Universal Robots PolyScope program: 20240830usb.urp

Program 20240830usb (installation=20240827 directory=/programs/Demos/usb createdIn=5.13.1 lastSavedIn=5.15.1 robotSerialNumber=20245500285)
Calibrated DH parameters: a=[0.000097, -0.210459, -0.026602, 0.000137, 0.000078, 0]; d=[0.162601, 254.180657, -54.076236, -199.970743, 0.099615, 0.099684]; alpha=[1.569796, -0.001455, 0.001957, 1.570525, -1.571561, 0]; deltaTheta=[0, -1.053331, 8.839472, -1.50296, 0.000002, 0]
InitVariablesNode
Robot Program (runOnlyOnce=false)
  MoveJ speed 60 deg/s, acceleration 80 deg/s^2 (useActiveTCP=true) feature=Base
    Waypoint 路点_2: TCP in base x=378.633 y=-400.967 z=269.032 mm, rx=0.8465 ry=2.3153 rz=-0.4134 rad; joints [111.319, -104.713, 126.879, -151.343, -75.69, 66.743] deg; TCP offset x=-0.17 y=0 z=192.95 mm, rx=0 ry=0 rz=0 rad
  Script: usb = rpc_factory("xmlrpc","http://192.168.1.7:9120/RPC2")
  SuppressedNode
    Script: usb.open()
  SuppressedNode
    Popup Message (haltProgram=false message=Grasp will close... inputType=Text)
  SuppressedNode
    Script: usb.close()
  Script: a=usb.get_target_pose()
  var_3 := p[0,0,0,0,0,0]
  Script: var_3[0] = -a[0]
  Script: var_3[2] = a[2]
  Script: var_3[4] = -a[4]
  Popup Message (haltProgram=false message=Get target pose. inputType=Variable) variable=var_3
  MoveJ speed 60 deg/s, acceleration 80 deg/s^2 (useActiveTCP=true) feature=Base
    Waypoint 路点_1: TCP in base x=381.086 y=-304.22 z=65.94 mm, rx=0 ry=3.0695 rz=-0.001 rad; joints [123.239, -85.086, 121.462, -128.728, -86.621, 33.467] deg; TCP offset x=-0.17 y=0 z=192.95 mm, rx=0 ry=0 rz=0 rad
  MoveJ speed 30 deg/s, acceleration 60 deg/s^2 (useActiveTCP=true) feature=Base
    var_1 := get_actual_tcp_pose()
    var_2 := pose_trans(var_1, var_3)
    MoveJ speed 60 deg/s, acceleration 80 deg/s^2 (useActiveTCP=true) feature=Base
      Waypoint Variable (Variable): motionParameters(jointSpeed=0.523599 jointAcceleration=1.047198 cartesianSpeed=0.25 cartesianAcceleration=1.2); variable(name=var_2)
  var_4 := var_2
  Script: var_4[2] = var_4[2] - 0.030
  MoveL speed 10 mm/s, acceleration 1200 mm/s^2 (useActiveTCP=true) feature=Base
    Waypoint Variable (Variable): variable(name=var_4)
    Popup Message (haltProgram=false message=Arrived! inputType=Text)
  Script: usb.open()
  Script: var_4[2] = var_4[2] + 0.008
  MoveL speed 10 mm/s, acceleration 1200 mm/s^2 (useActiveTCP=true) feature=Base
    Waypoint Variable (Variable): variable=var_4
  Script: usb.close()
  Script: var_4[2] = var_4[2] - 0.008
  MoveL speed 2 mm/s, acceleration 1000 mm/s^2 (useActiveTCP=true) feature=Base
    Waypoint Variable (Variable): variable=var_4
  Script: usb.open()
  Script: var_4[2] = var_4[2] + 0.04
  MoveL speed 30 mm/s, acceleration 500 mm/s^2 (useActiveTCP=true) feature=Base
    Waypoint Variable (Variable): variable=var_4
